//EL7201 | 1-chennel resolver terminal (ESS only use it for resolver input)
FUNCTION_BLOCK EL7201

VAR_INPUT
    En: BOOL;
    iTerminal_ID : INT;
    ErrorSystem : POINTER TO ST_ErrorSystem;
END_VAR

VAR_OUTPUT
    EnO: BOOL;
    bError: BOOL;
END_VAR

VAR
    //WC_State is handled by NC, so NOT included here.
    InfoData_State AT %I*: UINT;

    //FB-s
    EL7201_Error    : FB_TerminalError;
END_VAR

(*
* TODO: Test on hardware
*)

EnO:=En;

EL7201_Error(
    En := TRUE,
    iTerminal_ID := iTerminal_ID,
    bWcState := FALSE,
    uiInfoData_State := InfoData_State,
    pErrorSystem := ErrorSystem,
    bError => bError,
);

END_FUNCTION_BLOCK

(* stored: Version 1.1.0.1, ProductVersion 3.1.4024.0
   POU EL7201: Id {014d2d65-7ca8-4015-a842-40448ab49beb}, SpecialFunc None *)
